FUNCTION_BLOCK FB_SetAlarm
VAR_INPUT
	sMSg : STRING := '';
END_VAR
VAR_OUTPUT
END_VAR
VAR
END_VAR

GVL_HMI.o_bAlarmActive := TRUE;
GVL_HMI.o_sAlarmMessage := sMSg;

END_FUNCTION_BLOCK

(* stored: Version 1.1.0.1, ProductVersion 3.1.4024.6
   POU FB_SetAlarm: Id {3af222fe-3ae9-4d11-bf35-aa9ab617a18e}, SpecialFunc None *)
